# EPICS autosave request: LabJackApp/Db/LabJackWaveformGen_settings.req
$(P)WaveGenUserNumPoints
$(P)WaveGenIntNumPoints
$(P)WaveGenUserFrequency
$(P)WaveGenIntFrequency
$(P)WaveGenExtTrigger
$(P)WaveGenExtClock
$(P)WaveGenContinuous
